(* CoDeSys 2.3.9.50 project: 6C.pr6 *)
(* Libraries: STANDARD.LB6 5.6.98 12:03:02 *)

(* POU MAIN, LD *)
PROGRAM MAIN
VAR
	T1: TOF;
	C1: CTU;
	reset AT %IX0.7: BOOL;

	ACTUALTension AT %IX0.1: BOOL;
	EXTRATension AT %IX0.2: BOOL;
	Processon AT %QX0.4: BOOL;
	Start AT %IX0.0: BOOL;
	reducedThickness AT %QX0.0: BOOL;
	normalThickness AT %QX0.1: BOOL;
	IncreasedThickness AT %QX0.2: BOOL;
END_VAR
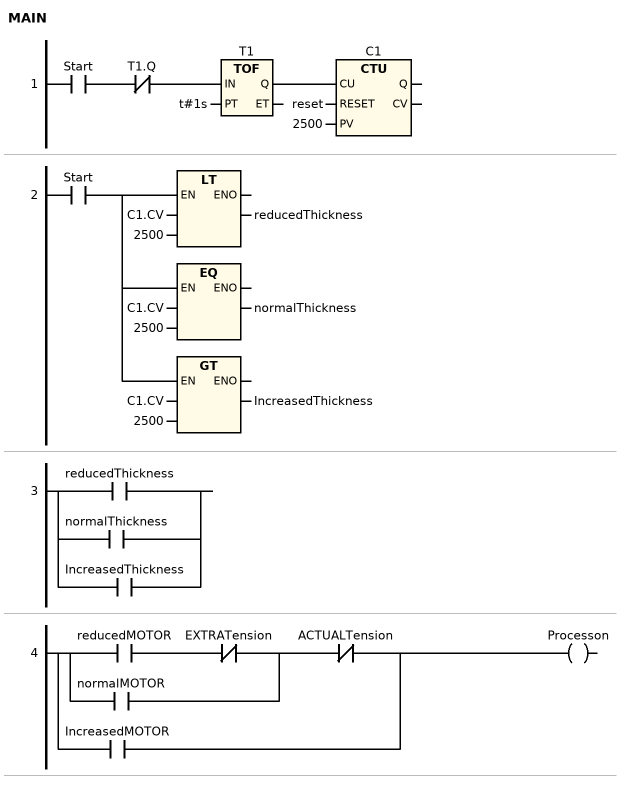
_LD_ (* Ladder Diagram *)
NETWORK 1
	[Start] - [/T1.Q] - T1:TOF(IN: *, PT: t#1s) - C1:CTU(CU: *, RESET: reset, PV: 2500)
NETWORK 2
	[Start]
		EN --- LT(C1.CV, 2500) => reducedThickness
		EN --- EQ(C1.CV, 2500) => normalThickness
		EN --- GT(C1.CV, 2500) => IncreasedThickness
NETWORK 3
	{ [reducedThickness] | [normalThickness] | [IncreasedThickness] }
NETWORK 4
	{ { [reducedMOTOR] - [/EXTRATension] | [normalMOTOR] } - [/ACTUALTension] | [IncreasedMOTOR] } --- (Processon)
_END_LD_
(* the same logic as Structured Text *)
(* Network 1 *)
T1(IN := Start AND NOT T1.Q, PT := t#1s);
C1(CU := T1.Q, RESET := reset, PV := 2500);
(* Network 2 *)
IF Start THEN
	reducedThickness := C1.CV < 2500;
	normalThickness := C1.CV = 2500;
	IncreasedThickness := C1.CV > 2500;
END_IF;
(* Network 3 *)
(* Network 4 *)
Processon := (reducedMOTOR AND NOT EXTRATension OR normalMOTOR) AND NOT ACTUALTension OR IncreasedMOTOR;
END_PROGRAM
